Omron CX-Programmer project 怴婯踢奂蕺改 (CX-Programmer 9.73)

# PLC 怴婯PC1: CJ1M CPU11

## Global symbols (name address type ; comment)
0.00 BOOL  ; 运转准备信号
0.01 BOOL  ; 手动/自动
0.02 BOOL  ; 复位
0.03 BOOL  ; 灯测试
0.04 BOOL  ; 拨码开关第5针
0.05 BOOL  ; 拨码开关第6针
0.06 BOOL  ; 拨码开关第9针
0.07 BOOL  ; 拨码开关第11针
0.08 BOOL  ; 保护罩闭合按钮
0.09 BOOL  ; 保护罩打开按钮
0.10 BOOL  ; 电机启动按钮
0.11 BOOL  ; 电机停止按钮
0.12 BOOL  ; 吸气按钮
0.13 BOOL  ; 吹气按钮
0.14 BOOL  ; 同步运行按钮
0.15 BOOL  ; 压力开关
1 CHANNEL  ; 初始位
11 CHANNEL  ; 位数
1.00 BOOL  ; 启动按钮
1.01 BOOL  ; 保护罩打开到位
1.02 BOOL  ; 保护罩闭合到位
1.15 BOOL  ; 工件放置
2.00 BOOL  ; 运转准备条件
2.01 BOOL  ; 运转准备灯
2.02 BOOL  ; 气源灯
2.03 BOOL  ; PC运行
2.04 BOOL  ; 原位灯
2.05 BOOL  ; 运转中灯
2.06 BOOL  ; LS异常灯
2.07 BOOL  ; 综合异常灯
2.08 BOOL  ; 蜂鸣器
2.09 BOOL  ; 保护罩闭合灯
2.10 BOOL  ; 保护罩打开灯
2.11 BOOL  ; 电机启动灯
2.12 BOOL  ; 电机停止灯
2.13 BOOL  ; 吹气灯
2.14 BOOL  ; 吸气灯
2.15 BOOL  ; 同步运行灯
3.00 BOOL  ; 保护罩闭合阀
3.01 BOOL  ; 保护罩打开阀
3.02 BOOL  ; 吹气阀
3.03 BOOL  ; 吸气阀
3.04 BOOL  ; 电机启动输出
H0.00 BOOL  ; 加工状态记忆
H20 CHANNEL  ; 加工数
T0000 BOOL  ; 手动转换稳定时间
T0001 BOOL  ; 自动转换稳定时间
T0002 BOOL  ; 非正常数码报警延时
T0003 BOOL  ; 半秒脉冲发生器1
T0004 BOOL  ; 半秒脉冲发生器2
T0011 BOOL  ; 同步时间延迟1
T0012 BOOL  ; 同步时间延迟2
T0013 BOOL  ; 同步时间延迟3
T0014 BOOL  ; 同步时间延迟4
T0015 BOOL  ; 同步时间延迟5
T0016 BOOL  ; 同步时间延迟6
T0020 BOOL  ; 自动启动稳定时间
T0021 BOOL  ; 吸气延时1
T0022 BOOL  ; 吸气延时2
T0023 BOOL  ; 吸气延时3
T0024 BOOL  ; 吸气延时4
T0025 BOOL  ; 吸气延时5
T0026 BOOL  ; 吸气延时6
T0030 BOOL  ; LS断电异常
T0031 BOOL  ; 动作异常报警
T0032 BOOL  ; LS得电异常
T0060 BOOL  ; 工件放置确认
T0061 BOOL  ; 工件取走确认
W0 CHANNEL  ; 数码
W0.00 BOOL  ; 运转准备有
W0.01 BOOL  ; 气源有
W0.02 BOOL  ; 原位置
W0.03 BOOL  ; 手动状态
W0.04 BOOL  ; 自动状态
W0.05 BOOL  ; 复位
W0.06 BOOL  ; 灯测试
W0.07 BOOL  ; 半秒脉冲
W10.00 BOOL  ; 保护罩手动闭合
W10.01 BOOL  ; 保护罩手动打开
W10.02 BOOL  ; 手动吹气
W10.03 BOOL  ; 手动吸气
W10.04 BOOL  ; 电机手动运转
W10.05 BOOL  ; 同步运行辅助
W10.06 BOOL  ; 同步运行启动脉冲
W10.07 BOOL  ; 同步运行停止
W11.01 BOOL  ; 同步时间1
W11.02 BOOL  ; 同步时间2
W11.03 BOOL  ; 同步时间3
W11.04 BOOL  ; 同步时间4
W11.05 BOOL  ; 同步时间5
W11.06 BOOL  ; 同步时间6
W20.00 BOOL  ; 自动启动脉冲
W20.01 BOOL  ; 第一步 闭合
W20.02 BOOL  ; 第二步 除尘
W20.03 BOOL  ; 第三步 打开
W20.04 BOOL  ; 工作完成信号
W20.05 BOOL  ; 自动运转中
W20.07 BOOL  ; 再启动防止
W30.00 BOOL  ; 自动启动条件
W30.01 BOOL  ; 工件未加工取走
W30.02 BOOL  ; 未取工件启动报警
W30.03 BOOL  ; 无工件启动报警
W3.01 BOOL  ; 非正常数码报警辅助
W3.02 BOOL  ; LS异常辅助
W3.10 BOOL  ; 综合异常辅助
W3.11 BOOL  ; 消声
W3.12 BOOL  ; 故障后回原位启动
W3.13 BOOL  ; 故障后回原位
W3.14 BOOL  ; 吸气延时辅助
W7 CHANNEL  ; 拨码开关
W7.01 BOOL  ; 数码1
W7.02 BOOL  ; 数码2
W7.03 BOOL  ; 数码3
W7.04 BOOL  ; 数码4
W7.05 BOOL  ; 数码5
W7.06 BOOL  ; 数码6

## Program 新程序1 (cyclic task 0)
; 项目介绍 / 1.	这个PLC程序实现了一个C3电枢异物吸引控制系统，应用于电机制造厂的电枢生产线，在电枢加工前通过吹气和吸气清除异物。 / 设备列表 / 1.	系统包含操作面板按钮，如运转准备信号按钮、手动/自动开关、保护罩闭合按钮、保护罩打开按钮、吹气按钮、吸气按钮等。 / 2.	系统还包括传感器，如工件放置传感器、保护罩闭合到位传感器、保护罩打开到位传感器，以及执行器，如保护罩闭合阀、保护罩打开阀、吹气阀、吸气阀。 / 3.	PLC系统使用CJ1M型号的CPU11，通过COM1端口通信。 / 代码思路 / 1.系统通过运转准备信号按钮启动，当运转准备灯亮起时，表示设备已就绪。 / 2.操作员可通过手动/自动切换开关选择模式，手动状态标志和自动状态标志通过定时器置位，确保模式切换稳定且唯一。 / 3.在手动模式下，操作员按下保护罩闭合按钮触发保护罩闭合阀，或按保护罩打开按钮触发保护罩打开阀，但两者不能同时动作，避免机械冲突。 / 4.吹气按钮和吸气按钮分别控制吹气阀和吸气阀，系统通过压力开关检测气源并点亮气源灯，但吹气和吸气动作当前未直接依赖气源状态。 / 5.在自动模式下，当工件放置传感器检测到电枢到位时，触发自动启动脉冲，经定时器确认后启动流程，需系统处于运转准备状态。 / 6.流程首先驱动保护罩闭合阀，此时需保护罩打开到位传感器为真，保证从打开状态开始闭合。 / 7.当保护罩闭合到位传感器确认闭合完成时，驱动吹气阀和吸气阀清除异物，但吹气和吸气动作当前未直接依赖气源状态。 / 8.清除完成后，驱动保护罩打开阀，需等待除尘完成且吹气和吸气停止。 / 9.整个过程中，保护罩状态由闭合到位传感器和打开到位传感器反馈，确保每一步安全过渡。 / 10.复位按钮可随时恢复初始状态，灯测试按钮用于检查所有指示灯（如气源灯、运转准备灯）是否正常。

### Section 主程序E_1_kenj_LOCALS_1_Temp_IDX

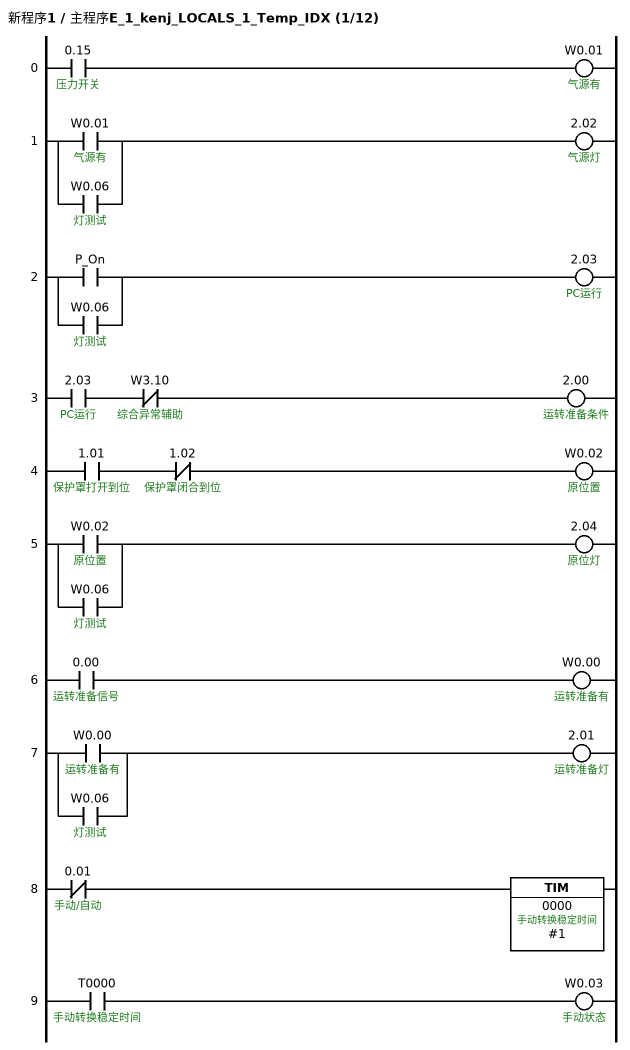
; rung 0
LD 0.15  ; 压力开关
OUT W0.01  ; 气源有
; rung 1
LD W0.01  ; 气源有
OR W0.06  ; 灯测试
OUT 2.02  ; 气源灯
; rung 2
LD P_On
OR W0.06  ; 灯测试
OUT 2.03  ; PC运行
; rung 3
LD 2.03  ; PC运行
ANDNOT W3.10  ; 综合异常辅助
OUT 2.00  ; 运转准备条件
; rung 4
LD 1.01  ; 保护罩打开到位
ANDNOT 1.02  ; 保护罩闭合到位
OUT W0.02  ; 原位置
; rung 5
LD W0.02  ; 原位置
OR W0.06  ; 灯测试
OUT 2.04  ; 原位灯
; rung 6
LD 0.00  ; 运转准备信号
OUT W0.00  ; 运转准备有
; rung 7
LD W0.00  ; 运转准备有
OR W0.06  ; 灯测试
OUT 2.01  ; 运转准备灯
; rung 8
LDNOT 0.01  ; 手动/自动
TIM 0000 #1  ; 手动转换稳定时间
; rung 9
LD T0000  ; 手动转换稳定时间
OUT W0.03  ; 手动状态

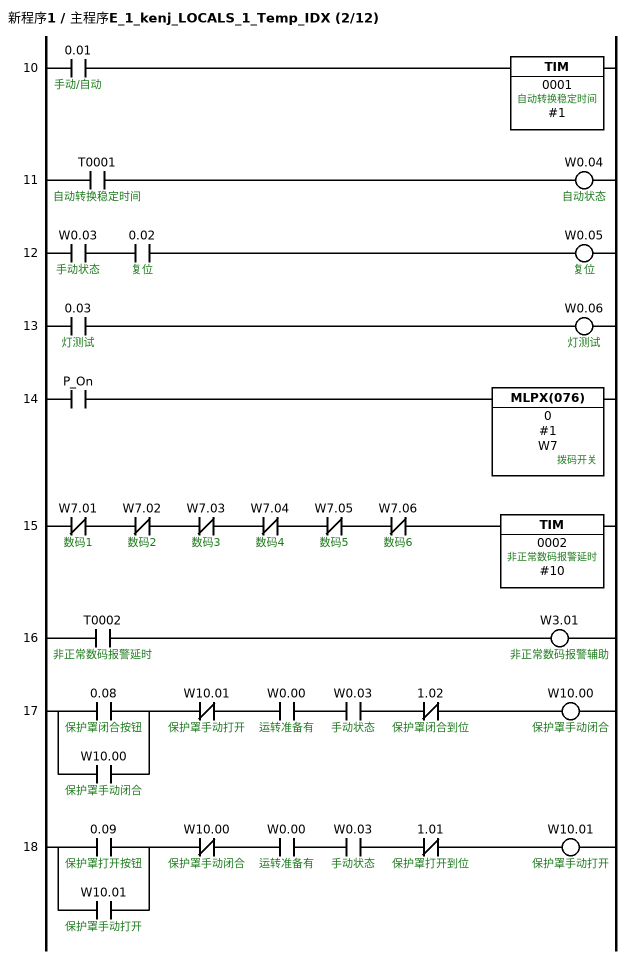
; rung 10
LD 0.01  ; 手动/自动
TIM 0001 #1  ; 自动转换稳定时间
; rung 11
LD T0001  ; 自动转换稳定时间
OUT W0.04  ; 自动状态
; rung 12
LD W0.03  ; 手动状态
AND 0.02  ; 复位
OUT W0.05  ; 复位
; rung 13
LD 0.03  ; 灯测试
OUT W0.06  ; 灯测试
; rung 14
LD P_On
MLPX(076) 0 #1 W7  ; 拨码开关  // 此命令有待试�
; rung 15
LDNOT W7.01  ; 数码1
ANDNOT W7.02  ; 数码2
ANDNOT W7.03  ; 数码3
ANDNOT W7.04  ; 数码4
ANDNOT W7.05  ; 数码5
ANDNOT W7.06  ; 数码6
TIM 0002 #10  ; 非正常数码报警延时
; rung 16
LD T0002  ; 非正常数码报警延时
OUT W3.01  ; 非正常数码报警辅助
; rung 17
LD 0.08  ; 保护罩闭合按钮
OR W10.00  ; 保护罩手动闭合
ANDNOT W10.01  ; 保护罩手动打开
AND W0.00  ; 运转准备有
AND W0.03  ; 手动状态
ANDNOT 1.02  ; 保护罩闭合到位
OUT W10.00  ; 保护罩手动闭合
; rung 18
LD 0.09  ; 保护罩打开按钮
OR W10.01  ; 保护罩手动打开
ANDNOT W10.00  ; 保护罩手动闭合
AND W0.00  ; 运转准备有
AND W0.03  ; 手动状态
ANDNOT 1.01  ; 保护罩打开到位
OUT W10.01  ; 保护罩手动打开

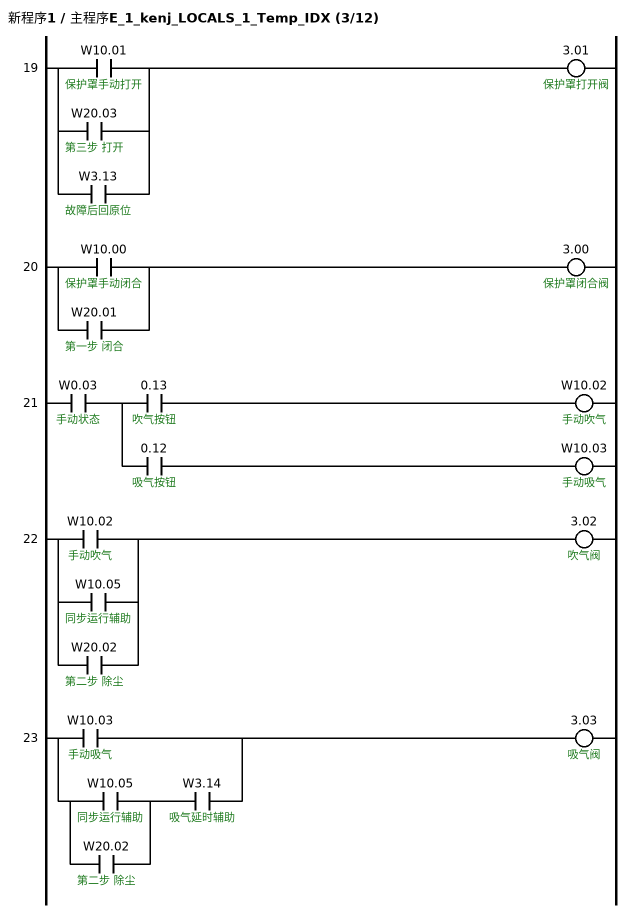
; rung 19
LD W10.01  ; 保护罩手动打开
OR W20.03  ; 第三步 打开
OR W3.13  ; 故障后回原位
OUT 3.01  ; 保护罩打开阀
; rung 20
LD W10.00  ; 保护罩手动闭合
OR W20.01  ; 第一步 闭合
OUT 3.00  ; 保护罩闭合阀
; rung 21
LD W0.03  ; 手动状态
OUT TR0
AND 0.13  ; 吹气按钮
OUT W10.02  ; 手动吹气
LD TR0
AND 0.12  ; 吸气按钮
OUT W10.03  ; 手动吸气
; rung 22
LD W10.02  ; 手动吹气
OR W10.05  ; 同步运行辅助
OR W20.02  ; 第二步 除尘
OUT 3.02  ; 吹气阀
; rung 23
LD W10.03  ; 手动吸气
LD W10.05  ; 同步运行辅助
OR W20.02  ; 第二步 除尘
AND W3.14  ; 吸气延时辅助
ORLD
OUT 3.03  ; 吸气阀

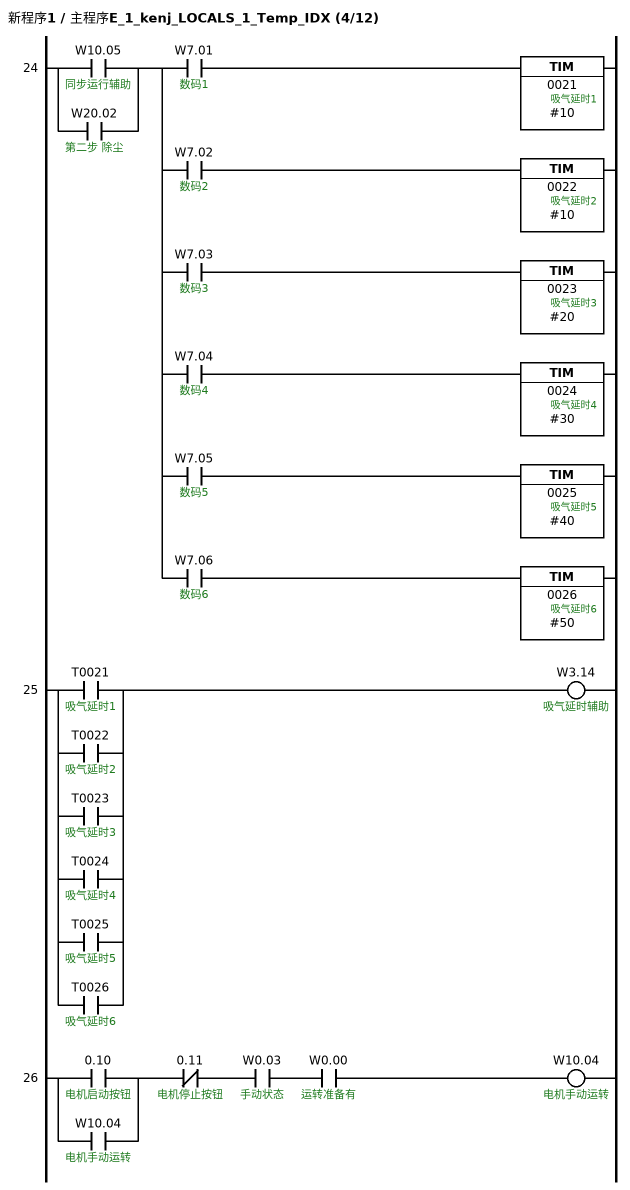
; rung 24
LD W10.05  ; 同步运行辅助
OR W20.02  ; 第二步 除尘
OUT TR0
AND W7.01  ; 数码1
TIM 0021 #10  ; 吸气延时1
LD TR0
AND W7.02  ; 数码2
TIM 0022 #10  ; 吸气延时2
LD TR0
AND W7.03  ; 数码3
TIM 0023 #20  ; 吸气延时3
LD TR0
AND W7.04  ; 数码4
TIM 0024 #30  ; 吸气延时4
LD TR0
AND W7.05  ; 数码5
TIM 0025 #40  ; 吸气延时5
LD TR0
AND W7.06  ; 数码6
TIM 0026 #50  ; 吸气延时6
; rung 25
LD T0021  ; 吸气延时1
OR T0022  ; 吸气延时2
OR T0023  ; 吸气延时3
OR T0024  ; 吸气延时4
OR T0025  ; 吸气延时5
OR T0026  ; 吸气延时6
OUT W3.14  ; 吸气延时辅助
; rung 26
LD 0.10  ; 电机启动按钮
OR W10.04  ; 电机手动运转
ANDNOT 0.11  ; 电机停止按钮
AND W0.03  ; 手动状态
AND W0.00  ; 运转准备有
OUT W10.04  ; 电机手动运转

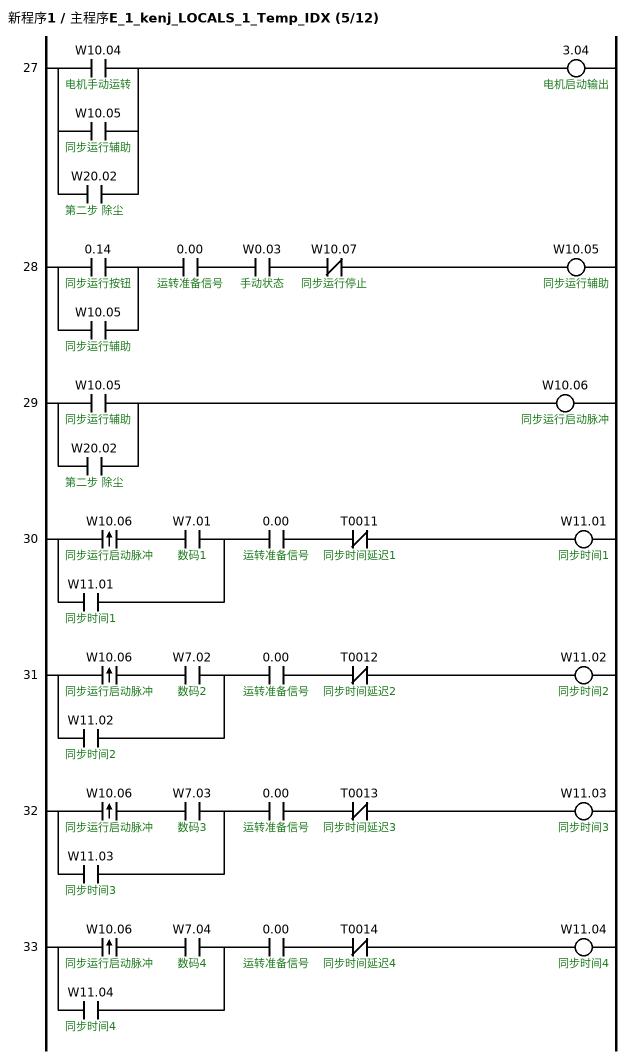
; rung 27
LD W10.04  ; 电机手动运转
OR W10.05  ; 同步运行辅助
OR W20.02  ; 第二步 除尘
OUT 3.04  ; 电机启动输出
; rung 28
LD 0.14  ; 同步运行按钮
OR W10.05  ; 同步运行辅助
AND 0.00  ; 运转准备信号
AND W0.03  ; 手动状态
ANDNOT W10.07  ; 同步运行停止
OUT W10.05  ; 同步运行辅助
; rung 29
LD W10.05  ; 同步运行辅助
OR W20.02  ; 第二步 除尘
OUT W10.06  ; 同步运行启动脉冲
; rung 30
@LD W10.06  ; 同步运行启动脉冲
AND W7.01  ; 数码1
OR W11.01  ; 同步时间1
AND 0.00  ; 运转准备信号
ANDNOT T0011  ; 同步时间延迟1
OUT W11.01  ; 同步时间1
; rung 31
@LD W10.06  ; 同步运行启动脉冲
AND W7.02  ; 数码2
OR W11.02  ; 同步时间2
AND 0.00  ; 运转准备信号
ANDNOT T0012  ; 同步时间延迟2
OUT W11.02  ; 同步时间2
; rung 32
@LD W10.06  ; 同步运行启动脉冲
AND W7.03  ; 数码3
OR W11.03  ; 同步时间3
AND 0.00  ; 运转准备信号
ANDNOT T0013  ; 同步时间延迟3
OUT W11.03  ; 同步时间3
; rung 33
@LD W10.06  ; 同步运行启动脉冲
AND W7.04  ; 数码4
OR W11.04  ; 同步时间4
AND 0.00  ; 运转准备信号
ANDNOT T0014  ; 同步时间延迟4
OUT W11.04  ; 同步时间4

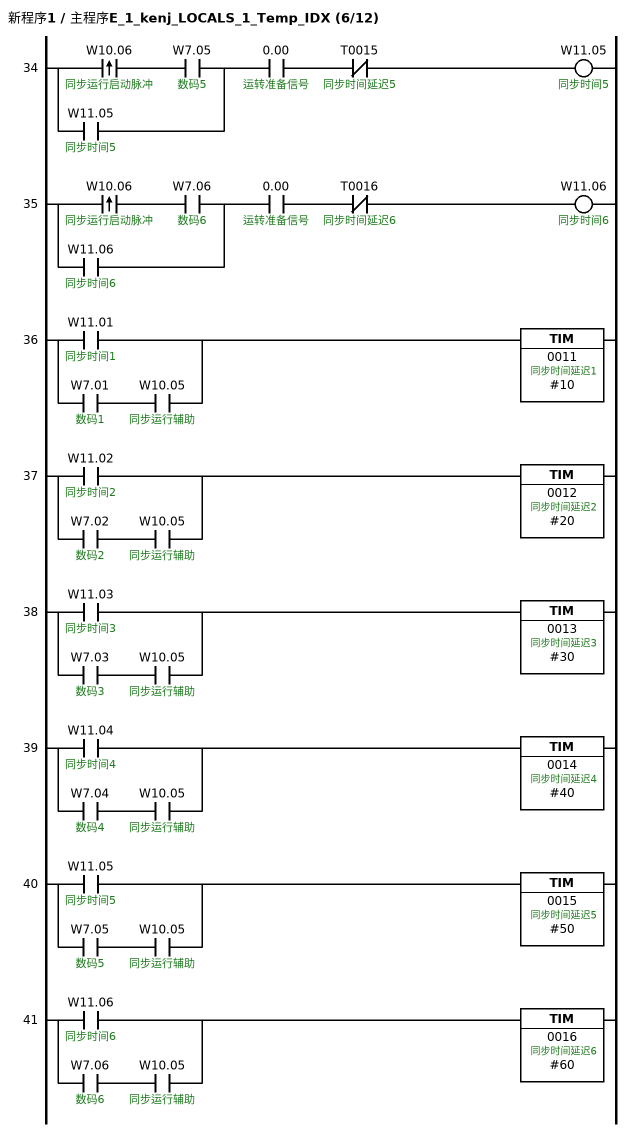
; rung 34
@LD W10.06  ; 同步运行启动脉冲
AND W7.05  ; 数码5
OR W11.05  ; 同步时间5
AND 0.00  ; 运转准备信号
ANDNOT T0015  ; 同步时间延迟5
OUT W11.05  ; 同步时间5
; rung 35
@LD W10.06  ; 同步运行启动脉冲
AND W7.06  ; 数码6
OR W11.06  ; 同步时间6
AND 0.00  ; 运转准备信号
ANDNOT T0016  ; 同步时间延迟6
OUT W11.06  ; 同步时间6
; rung 36
LD W11.01  ; 同步时间1
LD W7.01  ; 数码1
AND W10.05  ; 同步运行辅助
ORLD
TIM 0011 #10  ; 同步时间延迟1
; rung 37
LD W11.02  ; 同步时间2
LD W7.02  ; 数码2
AND W10.05  ; 同步运行辅助
ORLD
TIM 0012 #20  ; 同步时间延迟2
; rung 38
LD W11.03  ; 同步时间3
LD W7.03  ; 数码3
AND W10.05  ; 同步运行辅助
ORLD
TIM 0013 #30  ; 同步时间延迟3
; rung 39
LD W11.04  ; 同步时间4
LD W7.04  ; 数码4
AND W10.05  ; 同步运行辅助
ORLD
TIM 0014 #40  ; 同步时间延迟4
; rung 40
LD W11.05  ; 同步时间5
LD W7.05  ; 数码5
AND W10.05  ; 同步运行辅助
ORLD
TIM 0015 #50  ; 同步时间延迟5
; rung 41
LD W11.06  ; 同步时间6
LD W7.06  ; 数码6
AND W10.05  ; 同步运行辅助
ORLD
TIM 0016 #60  ; 同步时间延迟6

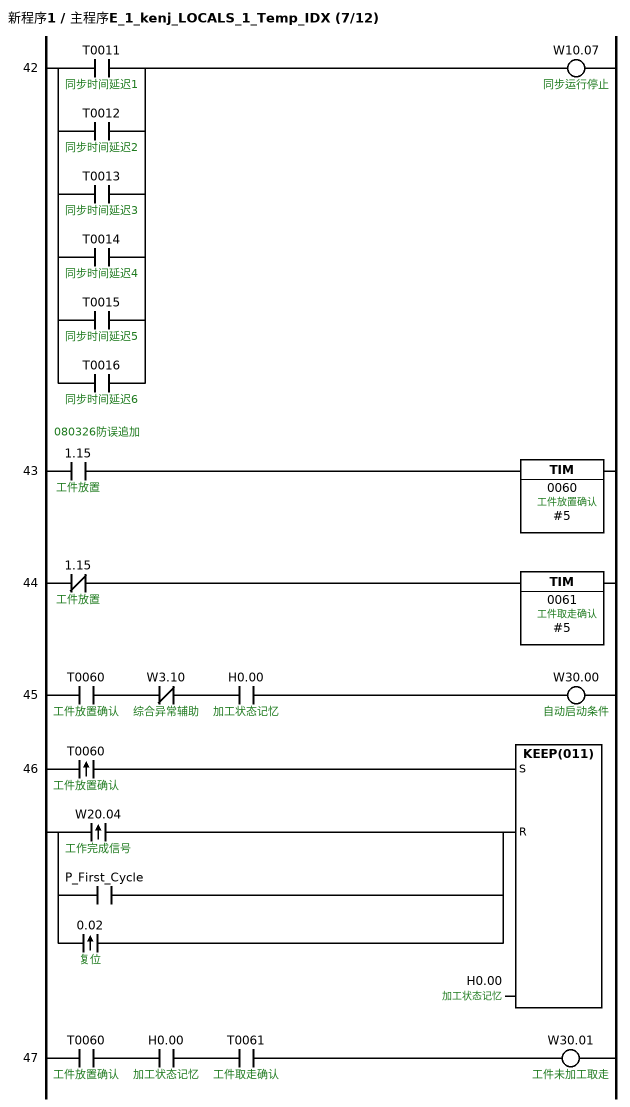
; rung 42
LD T0011  ; 同步时间延迟1
OR T0012  ; 同步时间延迟2
OR T0013  ; 同步时间延迟3
OR T0014  ; 同步时间延迟4
OR T0015  ; 同步时间延迟5
OR T0016  ; 同步时间延迟6
OUT W10.07  ; 同步运行停止
; rung 43: 080326防误追加
LD 1.15  ; 工件放置
TIM 0060 #5  ; 工件放置确认
; rung 44
LDNOT 1.15  ; 工件放置
TIM 0061 #5  ; 工件取走确认
; rung 45
LD T0060  ; 工件放置确认
ANDNOT W3.10  ; 综合异常辅助
AND H0.00  ; 加工状态记忆
OUT W30.00  ; 自动启动条件
; rung 46
@LD T0060  ; 工件放置确认
@LD W20.04  ; 工作完成信号
OR P_First_Cycle
@OR 0.02  ; 复位
KEEP(011) H0.00  ; 加工状态记忆
; rung 47
LD T0060  ; 工件放置确认
AND H0.00  ; 加工状态记忆
AND T0061  ; 工件取走确认
OUT W30.01  ; 工件未加工取走

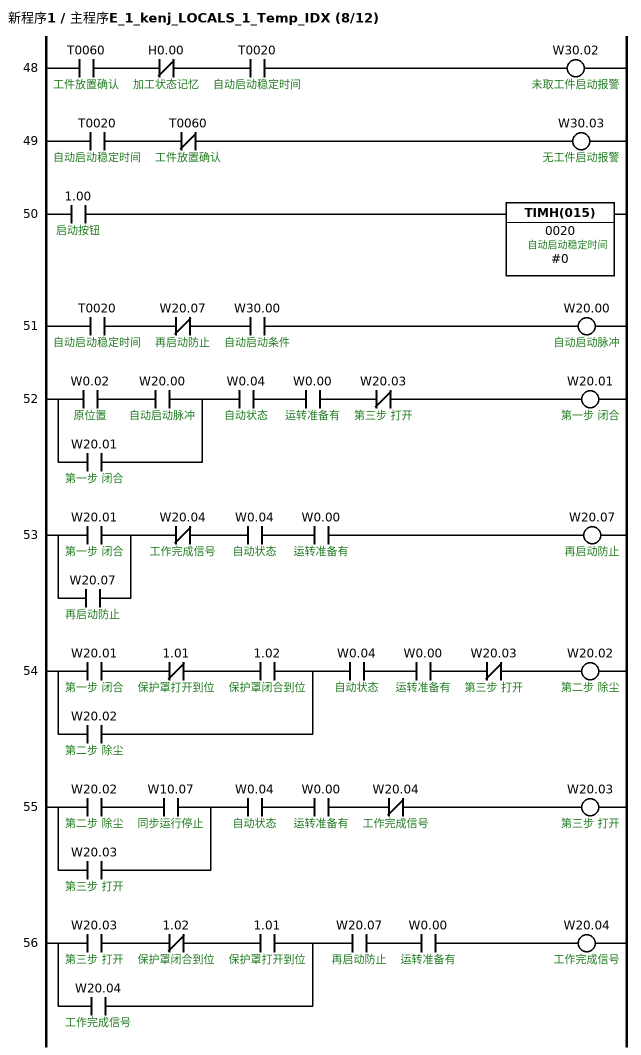
; rung 48
LD T0060  ; 工件放置确认
ANDNOT H0.00  ; 加工状态记忆
AND T0020  ; 自动启动稳定时间
OUT W30.02  ; 未取工件启动报警
; rung 49
LD T0020  ; 自动启动稳定时间
ANDNOT T0060  ; 工件放置确认
OUT W30.03  ; 无工件启动报警
; rung 50
LD 1.00  ; 启动按钮
TIMH(015) 0020 #0  ; 自动启动稳定时间
; rung 51
LD T0020  ; 自动启动稳定时间
ANDNOT W20.07  ; 再启动防止
AND W30.00  ; 自动启动条件
OUT W20.00  ; 自动启动脉冲
; rung 52
LD W0.02  ; 原位置
AND W20.00  ; 自动启动脉冲
OR W20.01  ; 第一步 闭合
AND W0.04  ; 自动状态
AND W0.00  ; 运转准备有
ANDNOT W20.03  ; 第三步 打开
OUT W20.01  ; 第一步 闭合
; rung 53
LD W20.01  ; 第一步 闭合
OR W20.07  ; 再启动防止
ANDNOT W20.04  ; 工作完成信号
AND W0.04  ; 自动状态
AND W0.00  ; 运转准备有
OUT W20.07  ; 再启动防止
; rung 54
LD W20.01  ; 第一步 闭合
ANDNOT 1.01  ; 保护罩打开到位
AND 1.02  ; 保护罩闭合到位
OR W20.02  ; 第二步 除尘
AND W0.04  ; 自动状态
AND W0.00  ; 运转准备有
ANDNOT W20.03  ; 第三步 打开
OUT W20.02  ; 第二步 除尘
; rung 55
LD W20.02  ; 第二步 除尘
AND W10.07  ; 同步运行停止
OR W20.03  ; 第三步 打开
AND W0.04  ; 自动状态
AND W0.00  ; 运转准备有
ANDNOT W20.04  ; 工作完成信号
OUT W20.03  ; 第三步 打开
; rung 56
LD W20.03  ; 第三步 打开
ANDNOT 1.02  ; 保护罩闭合到位
AND 1.01  ; 保护罩打开到位
OR W20.04  ; 工作完成信号
AND W20.07  ; 再启动防止
AND W0.00  ; 运转准备有
OUT W20.04  ; 工作完成信号

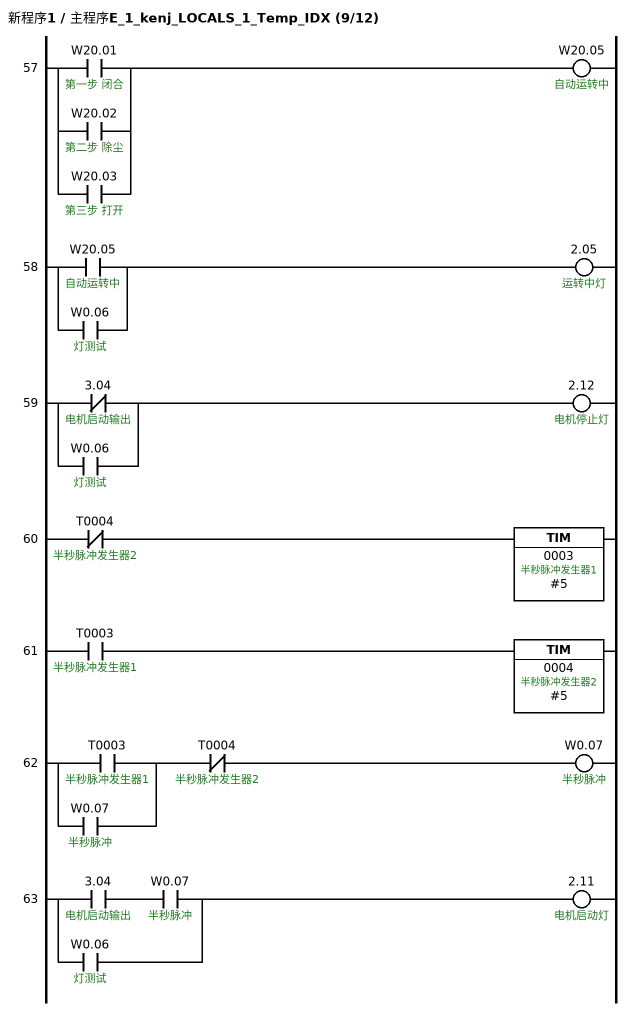
; rung 57
LD W20.01  ; 第一步 闭合
OR W20.02  ; 第二步 除尘
OR W20.03  ; 第三步 打开
OUT W20.05  ; 自动运转中
; rung 58
LD W20.05  ; 自动运转中
OR W0.06  ; 灯测试
OUT 2.05  ; 运转中灯
; rung 59
LDNOT 3.04  ; 电机启动输出
OR W0.06  ; 灯测试
OUT 2.12  ; 电机停止灯
; rung 60
LDNOT T0004  ; 半秒脉冲发生器2
TIM 0003 #5  ; 半秒脉冲发生器1
; rung 61
LD T0003  ; 半秒脉冲发生器1
TIM 0004 #5  ; 半秒脉冲发生器2
; rung 62
LD T0003  ; 半秒脉冲发生器1
OR W0.07  ; 半秒脉冲
ANDNOT T0004  ; 半秒脉冲发生器2
OUT W0.07  ; 半秒脉冲
; rung 63
LD 3.04  ; 电机启动输出
AND W0.07  ; 半秒脉冲
OR W0.06  ; 灯测试
OUT 2.11  ; 电机启动灯

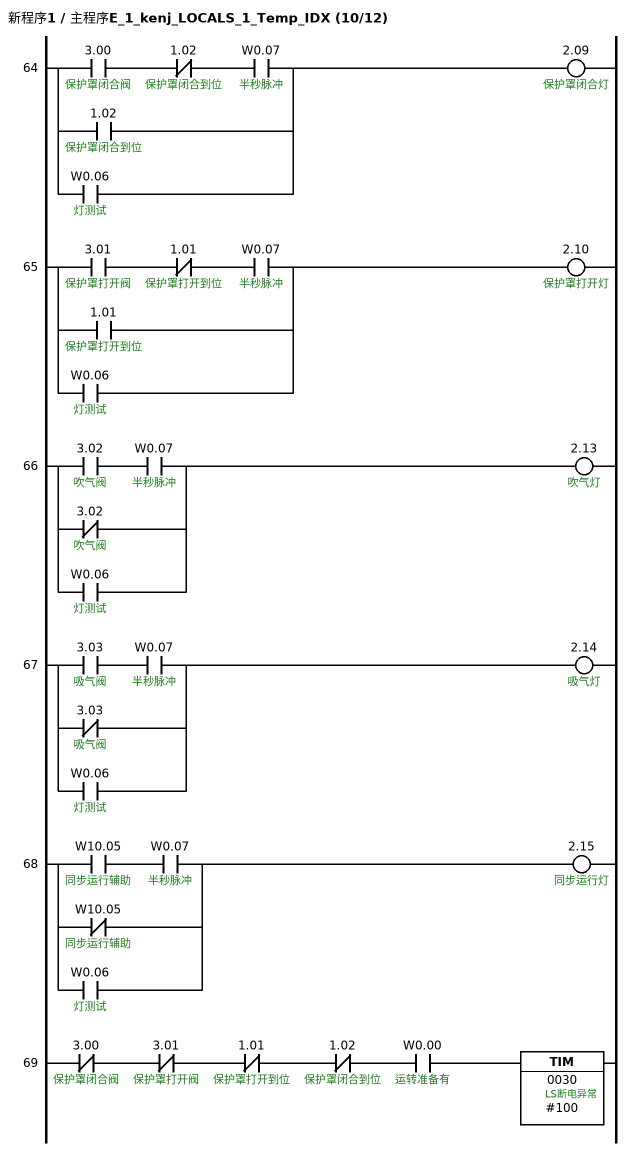
; rung 64
LD 3.00  ; 保护罩闭合阀
ANDNOT 1.02  ; 保护罩闭合到位
AND W0.07  ; 半秒脉冲
OR 1.02  ; 保护罩闭合到位
OR W0.06  ; 灯测试
OUT 2.09  ; 保护罩闭合灯
; rung 65
LD 3.01  ; 保护罩打开阀
ANDNOT 1.01  ; 保护罩打开到位
AND W0.07  ; 半秒脉冲
OR 1.01  ; 保护罩打开到位
OR W0.06  ; 灯测试
OUT 2.10  ; 保护罩打开灯
; rung 66
LD 3.02  ; 吹气阀
AND W0.07  ; 半秒脉冲
ORNOT 3.02  ; 吹气阀
OR W0.06  ; 灯测试
OUT 2.13  ; 吹气灯
; rung 67
LD 3.03  ; 吸气阀
AND W0.07  ; 半秒脉冲
ORNOT 3.03  ; 吸气阀
OR W0.06  ; 灯测试
OUT 2.14  ; 吸气灯
; rung 68
LD W10.05  ; 同步运行辅助
AND W0.07  ; 半秒脉冲
ORNOT W10.05  ; 同步运行辅助
OR W0.06  ; 灯测试
OUT 2.15  ; 同步运行灯
; rung 69
LDNOT 3.00  ; 保护罩闭合阀
ANDNOT 3.01  ; 保护罩打开阀
ANDNOT 1.01  ; 保护罩打开到位
ANDNOT 1.02  ; 保护罩闭合到位
AND W0.00  ; 运转准备有
TIM 0030 #100  ; LS断电异常

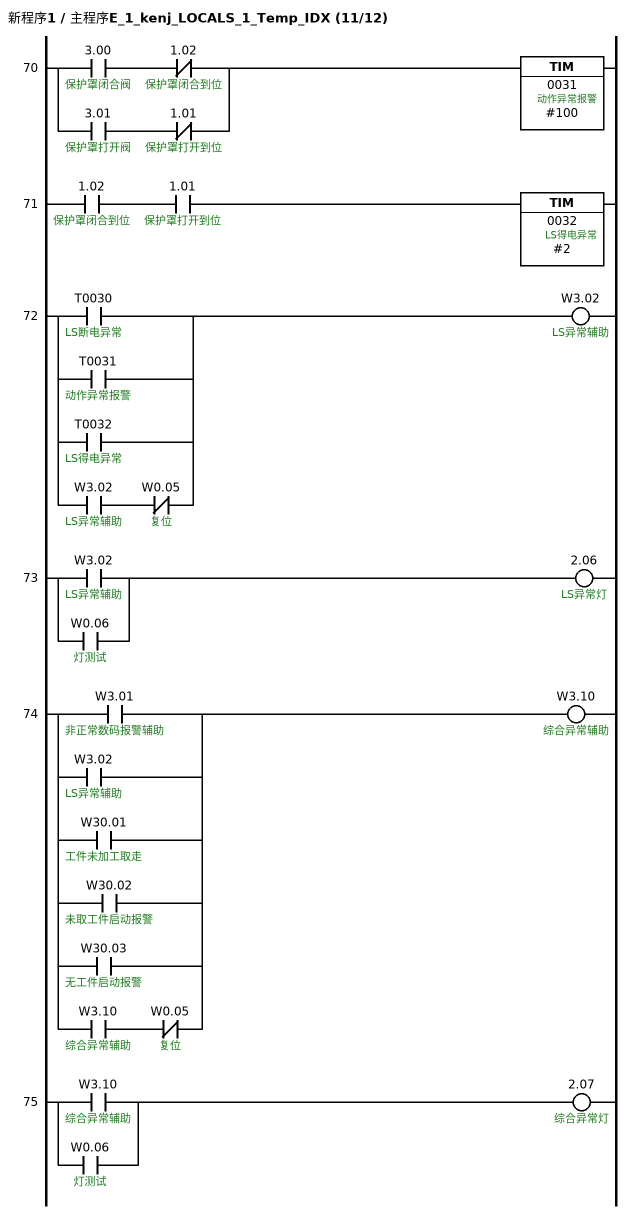
; rung 70
LD 3.00  ; 保护罩闭合阀
ANDNOT 1.02  ; 保护罩闭合到位
LD 3.01  ; 保护罩打开阀
ANDNOT 1.01  ; 保护罩打开到位
ORLD
TIM 0031 #100  ; 动作异常报警
; rung 71
LD 1.02  ; 保护罩闭合到位
AND 1.01  ; 保护罩打开到位
TIM 0032 #2  ; LS得电异常
; rung 72
LD T0030  ; LS断电异常
OR T0031  ; 动作异常报警
OR T0032  ; LS得电异常
LD W3.02  ; LS异常辅助
ANDNOT W0.05  ; 复位
ORLD
OUT W3.02  ; LS异常辅助
; rung 73
LD W3.02  ; LS异常辅助
OR W0.06  ; 灯测试
OUT 2.06  ; LS异常灯
; rung 74
LD W3.01  ; 非正常数码报警辅助
OR W3.02  ; LS异常辅助
OR W30.01  ; 工件未加工取走
OR W30.02  ; 未取工件启动报警
OR W30.03  ; 无工件启动报警
LD W3.10  ; 综合异常辅助
ANDNOT W0.05  ; 复位
ORLD
OUT W3.10  ; 综合异常辅助
; rung 75
LD W3.10  ; 综合异常辅助
OR W0.06  ; 灯测试
OUT 2.07  ; 综合异常灯

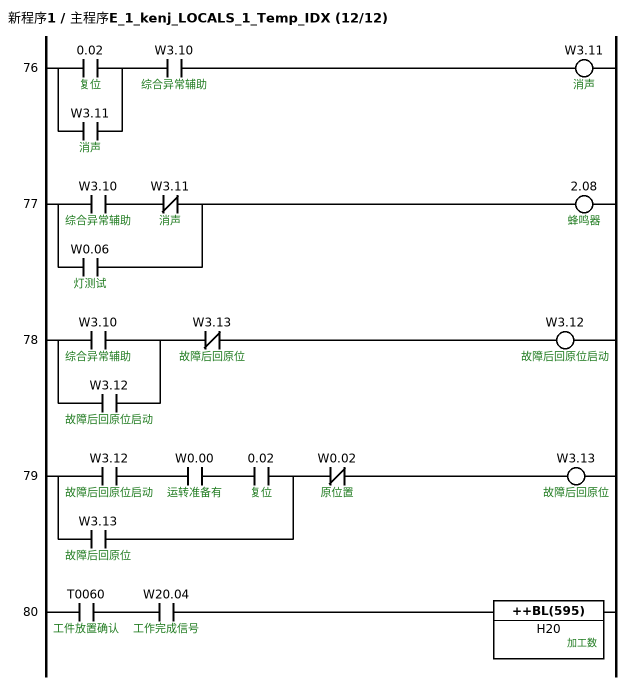
; rung 76
LD 0.02  ; 复位
OR W3.11  ; 消声
AND W3.10  ; 综合异常辅助
OUT W3.11  ; 消声
; rung 77
LD W3.10  ; 综合异常辅助
ANDNOT W3.11  ; 消声
OR W0.06  ; 灯测试
OUT 2.08  ; 蜂鸣器
; rung 78
LD W3.10  ; 综合异常辅助
OR W3.12  ; 故障后回原位启动
ANDNOT W3.13  ; 故障后回原位
OUT W3.12  ; 故障后回原位启动
; rung 79
LD W3.12  ; 故障后回原位启动
AND W0.00  ; 运转准备有
AND 0.02  ; 复位
OR W3.13  ; 故障后回原位
ANDNOT W0.02  ; 原位置
OUT W3.13  ; 故障后回原位
; rung 80
LD T0060  ; 工件放置确认
AND W20.04  ; 工作完成信号
++BL(595) H20  ; 加工数

### Section END
; rung 0
END(001)